FUNCTION_BLOCK FB_RobotArm
VAR
	Inputs 	AT%I* 	: ST_Inputs;
	Outputs AT%Q* 	: ST_Outputs;
	RobotArmJoints 	: ARRAY [1..GVL_RobotArm.NUMBER_OF_JOINTS] OF INT;
	Index 			: INT;
	JointTurnStep	: INT;
	
	//BoxPlaceLocation	: ARRAY [E_BoxPlaceDirection.PLACE1..E_BoxPlaceDirection.LastPlace] OF INT;
END_VAR

VAR PERSISTENT
	LSTEPS		: INT := 0;
	RSTEPS		: INT := 0;
	FirstScan 	: BOOL := TRUE;	
	
	InputsDecoupled		: ST_Inputs;
END_VAR

_M_StatusUpdate();


(*
	WRITE PUBLIC METHODS TO DO THE FOLLOWING:
	MOVE ONLY
		1. Move hand to Place #1
		2. Move hand to Place #2
		
	MOVE + GRIP																//Why did you decide to ad Move in the method?
		3. PickUpFromPlace( placenum := x )
		4. PlaceTo( placenum := x )

*)

METHOD PRIVATE _M_DefaultPosition : BOOL
VAR
	Index		: INT;
END_VAR
_M_GripControl( Close := TRUE ); // METHOD( INPUT := , OUTPUT => )
	
FOR Index := 1 TO GVL_RobotArm.NUMBER_OF_JOINTS DO 
	Outputs.JOINT_TURN_LEFT[Index]	:=	FALSE;
	Outputs.JOINT_TURN_RIGHT[Index]	:=	FALSE;//optimisation of//inputs.JOINT_TURN_RIGHT1:=inputs.JOINT_TURN_RIGHT2:=inputs.JOINT_TURN_RIGHT3:=inputs.JOINT_TURN_RIGHT4:=FALSE;
	LSTEPS:=RSTEPS:=0; 
END_FOR
END_METHOD

METHOD PRIVATE _M_GripControl : BOOL
VAR_INPUT
	Close	: BOOL;
END_VAR
	Outputs.GRIP_CLOSE := Close;
Outputs.GRIP_OPEN := NOT Close;
END_METHOD

METHOD PRIVATE _M_StatusUpdate : BOOL
VAR_INPUT
END_VAR
InputsDecoupled.GRIP_CONDITION := Inputs.GRIP_CONDITION; 

FOR Index := 1 TO GVL_RobotArm.NUMBER_OF_JOINTS DO
	InputsDecoupled.JOINT_LEFT_SIGNAL[Index] := Inputs.JOINT_LEFT_SIGNAL[Index];
	InputsDecoupled.JOINT_RIGHT_SIGNAL[Index] := Inputs.JOINT_RIGHT_SIGNAL[Index];
END_FOR

InputsDecoupled.PLACE1 := Inputs.PLACE1;
InputsDecoupled.PLACE2 := Inputs.PLACE2;
END_METHOD

METHOD PRIVATE _M_StraightJoint : BOOL
VAR
	Joint				: INT :=1;
END_VAR
Outputs.GRIP_CLOSE:=TRUE;

Outputs.JOINT_TURN_LEFT[Joint] := FALSE;
Outputs.JOINT_TURN_RIGHT[Joint] := FALSE;

//FOR Index := 1 TO GVL_RobotArm.NUMBER_OF_JOINTS BY 1 DO
//	Outputs.JOINT_TURN_LEFT	[Index]:=FALSE;
//	Outputs.JOINT_TURN_RIGHT_RIGHT	[Index]:=FALSE;
//END_FOR

(* CASE StraightPosition OF 
1:	inputs.JOINT_TURN_LEFT1:=FALSE;
	inputs.JOINT_TURN_RIGHT1:=FALSE;
2: 	inputs.JOINT_TURN_LEFT2:=FALSE;
	inputs.JOINT_TURN_RIGHT2:=FALSE;
3: 	inputs.JOINT_TURN_LEFT3:=FALSE;
	inputs.JOINT_TURN_RIGHT3:=FALSE;
4: 	inputs.JOINT_TURN_LEFT4:=FALSE;
	inputs.JOINT_TURN_RIGHT4:=FALSE;	
END_CASE *)
END_METHOD

METHOD PUBLIC M_MoveToPlace1 : BOOL
VAR	
END_VAR
_M_DefaultPosition();

//Inputs.GRIP_CONDITION := FALSE;

//M_TurnJoint( TurnDirection := E_RobotArmJointDirection.LEFT, Joint := Index); (*Not clear how use enumeration / for example, can I write  - E_RobotArmJointDirection.1*)
//M_TurnJoint (TurnDirection := E_BoxPlaceDirection.PLACE1 , E_RobotArmJointDirection.LEFT); // which line is correct in that case?

//FOR Index := 1 TO GVL_RobotArm.NUMBER_OF_JOINTS DO
//	M_TurnJoint( TurnDirection := E_RobotArmJointDirection.LEFT, Joint := Index );
//END_FOR

CASE JointTurnStep OF
	1:
		M_TurnJoint( TurnDirection := E_RobotArmJointDirection.LEFT, Joint := JointTurnStep );
		IF InputsDecoupled.JOINT_LEFT_SIGNAL[JointTurnStep] THEN
			JointTurnStep := 2;
		END_IF
	2: 
		M_TurnJoint( TurnDirection := E_RobotArmJointDirection.LEFT, Joint := JointTurnStep );
		IF InputsDecoupled.JOINT_LEFT_SIGNAL[JointTurnStep] THEN
			JointTurnStep := 3;
		END_IF
	3: 
		M_TurnJoint( TurnDirection := E_RobotArmJointDirection.LEFT, Joint := JointTurnStep );
		IF InputsDecoupled.JOINT_LEFT_SIGNAL[JointTurnStep] THEN
			M_PickUpFromThePlace.PLACE_NUM	:=1;
		END_IF
END_CASE




(*

	1. Return to default position 
	2. Move hand to Place 1
	3. Open Grip 
	...
	optionally: return to default position BUT returning to default must be performed ONLY IF GRIP_CONDITION EMPTY


_M_DefaultPosition(Default:=TRUE);
M_TurnJoint(TurnDirection:='LEFT');
outputs.GRIP_OPEN:=FALSE;

IF Inputs.GRIP_CONDITION THEN
	inputs.GRIP_CONDITION:=FALSE;
 _M_DefaultPosition(Default:=TRUE);

END_IF
*)
END_METHOD

METHOD PUBLIC M_MoveToPlace2 : BOOL
VAR
END_VAR


CASE JointTurnStep OF
	1:
		M_TurnJoint( TurnDirection := E_RobotArmJointDirection.RIGHT, Joint := JointTurnStep );
		IF InputsDecoupled.JOINT_RIGHT_SIGNAL[JointTurnStep] THEN
			JointTurnStep := 2;
		END_IF
	2: 
		M_TurnJoint( TurnDirection := E_RobotArmJointDirection.RIGHT, Joint := JointTurnStep );
		IF InputsDecoupled.JOINT_RIGHT_SIGNAL[JointTurnStep] THEN
			JointTurnStep := 3;
		END_IF
	3: 
		M_TurnJoint( TurnDirection := E_RobotArmJointDirection.RIGHT, Joint := JointTurnStep );
		IF InputsDecoupled.JOINT_RIGHT_SIGNAL[JointTurnStep] THEN
			M_PlaceTo.PLACE_NUM	:=2;
		END_IF
END_CASE





(*

	1. Return to default position 
	2. Move hand to Place 2
	3. Open Grip
	...
	optionally: return to default position BUT returning to default must be performed ONLY IF GRIP_CONDITION EMPTY

*)

//_M_DefaultPosition(Default:=TRUE);
//M_TurnJoint(TurnDirection:='RIGHT');
//outputs.GRIP_OPEN:=TRUE;

//IF outputs.GRIP_OPEN THEN
//	inputs.GRIP_CONDITION:=FALSE;
// _M_DefaultPosition(Default:=TRUE);

//END_IF
END_METHOD

METHOD PUBLIC M_PickUpFromThePlace : BOOL
VAR_INPUT
	PLACE_NUM : INT;
END_VAR
(*

	1. Return to default position 
	2. Move hand to Place 1
	3. Open Grip
	4. Close Grip when picked up (picked up => GRIP_CONDITION = TRUE)
	...
	optionally: return to default position

*)

CASE PLACE_NUM OF
	
	1: // pick from place 1
	_M_DefaultPosition();		
	M_MoveToPlace1();
	_M_GripControl(Close :=	 TRUE);
		
	2: // pick from place 2
	_M_DefaultPosition();		
	M_MoveToPlace2();
	_M_GripControl(Close :=	 TRUE);
	
END_CASE

(*
_M_DefaultPosition();
M_MoveToPlace1();
IF inputs.PLACE1 THEN
	Inputs.GRIP_CONDITION	:=	FALSE;
	_M_GripControl(Close	:=	FALSE);
ELSIF Inputs.GRIP_CONDITION	THEN
	Outputs.GRIP_CLOSE		:=TRUE;
	_M_DefaultPosition();
IF inputs.GRIP_CONDITION:=TRUE AND inputs.PLACE1:=FALSE THEN
	_M_DefaultPosition();
END_IF
END_IF
*)

//IF outputs.GRIP_OPEN THEN
//	outputs.GRIP_CLOSE		:=FALSE;
//	inputs.PLACE1			:=TRUE;
//	inputs.GRIP_CONDITION	:=FALSE;
//ELSIF inputs.GRIP_CONDITION THEN
//	Outputs.GRIP_CLOSE		:=TRUE;
//	_M_DefaultPosition();
//END_IF
END_METHOD

METHOD PUBLIC M_PlaceTo : BOOL
VAR_INPUT
	PLACE_NUM : INT;
END_VAR
(*

	1. Return to default position 
	2. Move hand to Place 2
	3. Open Grip
	4. Close Grip when picked up (picked up => GRIP_CONDITION = TRUE)
	...
	optionally: return to default position

*)

CASE PLACE_NUM OF
	1:
	_M_DefaultPosition();
	M_MoveToPlace1();	
	_M_GripControl(Close :=	 FALSE);
		
	2:
	_M_DefaultPosition();
	M_MoveToPlace2();
	_M_GripControl(Close :=	 FALSE);
	
END_CASE




//_M_DefaultPosition(Default:=TRUE);
//M_TurnJoint(TurnDirection:='RIGHT');
//IF inputs.GRIP_CONDITION THEN
//	outputs.GRIP_OPEN		:=TRUE;
//	inputs.PLACE2			:=FALSE;
//ELSIF inputs.GRIP_CONDITION:=FALSE THEN
//	_M_DefaultPosition(Default:=TRUE);
//END_IF
END_METHOD

METHOD PUBLIC M_TurnJoint : BOOL
VAR_INPUT
	TurnDirection 	: INT; // left / right
	Joint			: INT; // 1..GVL_RobotArm.MAX_JOINT
END_VAR
//_M_StraightJoint(); // Is it correct line?
CASE TurnDirection OF 
	E_RobotArmJointDirection.LEFT:// turn left  // ( Style of writing?)
		Outputs.JOINT_TURN_LEFT[Joint] := TRUE;
	E_RobotArmJointDirection.RIGHT: // turn right
		Outputs.JOINT_TURN_RIGHT[Joint] := TRUE;
END_CASE
END_METHOD

END_FUNCTION_BLOCK

(* stored: Version 1.1.0.1, ProductVersion 3.1.4024.9
   POU FB_RobotArm: Id {791aebaa-e1af-4e34-82e6-21b6dcafec81}, SpecialFunc None
   Folder Private: Id {8e206af4-6c72-4040-98dd-746c939058b7}
   Method _M_DefaultPosition: Id {b4076654-83fc-4691-b1b5-978eda6f60b7}
   Method _M_GripControl: Id {4500713e-daab-4b5f-93b1-f1dfd3fbfba4}
   Method _M_StatusUpdate: Id {424b32d3-2991-4e75-a053-29a008bea2c1}
   Method _M_StraightJoint: Id {3a826016-47df-4ee5-b177-5499df6b2db5}
   Method M_MoveToPlace1: Id {7a23719a-1aae-4640-a5ff-01800871be7e}
   Method M_MoveToPlace2: Id {0e169f60-7ed8-4039-bfcf-3f2af81e03a2}
   Method M_PickUpFromThePlace: Id {bb47bc22-22d9-491b-a40c-674ad464a234}
   Method M_PlaceTo: Id {9e7cd9ea-bfbb-4743-ac1e-c348e4a0ec1b}
   Method M_TurnJoint: Id {215986a3-b2d9-4a5b-a2c6-326f10567f86} *)
